INTERFACE I_Override EXTENDS I_Base

{attribute 'monitoring' := 'call'}
PROPERTY Override : LREAL
SET
END_SET
END_PROPERTY

END_INTERFACE

(* stored: Version 1.1.0.1, ProductVersion 3.1.4026.18
   Itf I_Override: Id {079ec021-667a-4390-bf30-3cf6bc7f151f}
   Property Override: Id {5c3080d9-496b-4ed4-8bd6-19dfd5da33c2}
   Set Set: Id {a89271c7-ac3a-48aa-8737-188977c54c23} *)
